// TIA Portal V17 export
// export: Created 2024-06-14T09:52:51.242704Z, ExportSetting WithDefaults, DisplayName Totally Integrated Automation Portal, DisplayVersion V17, DisplayName TIA Portal Openness, DisplayVersion V17, DisplayName TIA Portal Version Control Interface, DisplayVersion V17, DisplayName Simotion SCOUT TIA, DisplayVersion 5.4.3.0, DisplayName SINAMICS Startdrive Advanced, DisplayVersion V17 SP1 Update 1, DisplayName SINAMICS Startdrive G110M, G120, G120C, G120D, G120P, G115D, DisplayVersion V17 SP1 Update 1, DisplayName SINAMICS Startdrive G130, G150, S120, S150, SINAMICS MV, S210, DisplayVersion V17 SP1 Update 1, DisplayName STEP 7 Professional, DisplayVersion V17, DisplayName STEP 7 Safety, DisplayVersion V17, DisplayName WinCC Professional, DisplayVersion V17
DATA_BLOCK "MASTER_SETUP_DB"   // DB13
{ S7_Optimized_Access := 'FALSE' }
VERSION : 0.1
// stored: AutoNumber true, DBAccessibleFromOPCUA true, IsOnlyStoredInLoadMemory false, IsWriteProtectedInAS false
   VAR RETAIN
      Enable_Station1 : Bool;
      Enable_Station4 : Bool;
      S1_Enabled_Station : Array[1..6] of Bool;
      S4_Enabled_Station : Array[1..6] of Bool;
      S1_Total_Station : Int;
      S4_Total_Station : Int;
      Enabled_Station_S1 : Int;
      Enabled_Station_S4 : Int;
      Enabled_Station_S5 : Int;
      S5_Enabled_Station : Array[1..6] of Bool;
      S5_Total_Station : Int;
      Enable_Station5 : Bool;
   END_VAR
BEGIN
END_DATA_BLOCK
